{attribute 'TcRpcEnable'}
FUNCTION_BLOCK GetTc3Licenses IMPLEMENTS I_GetTc3Licenses
VAR_INPUT
END_VAR
VAR_OUTPUT
END_VAR
VAR
END_VAR
VAR
    // Internal
    fbGetLicensesEx : FB_GetLicensesEx;
    stAllLicensesInfos : ST_AllLicensesInfos;
    
    _sNetId   : T_AmsNetId;
    
    _fbJson         : FB_JsonSaxWriter;
    _fbJsonDataType : FB_JsonReadWriteDataType;
    
END_VAR
VAR
    stInfoData : ST_LicenseDetailsSmall;
    sReturn : STRING(30_000);
END_VAR


// include: Tc2_Utilities
// Realtime -> Global Max Stack = 2048kb

{attribute 'monitoring' := 'call'}
PROPERTY CountDemoLicenses : UDINT
GET

CountDemoLicenses := stAllLicensesInfos.DemoLicenses.Count;
END_GET
END_PROPERTY

{attribute 'monitoring' := 'call'}
PROPERTY CountFailedLicenses : UDINT
GET

CountFailedLicenses := stAllLicensesInfos.FailedLicenses.Count;
END_GET
END_PROPERTY

{attribute 'monitoring' := 'call'}
PROPERTY CountInvalidLicenses : UDINT
GET

CountInvalidLicenses := stAllLicensesInfos.InvalidLicenses.Count;
END_GET
END_PROPERTY

{attribute 'monitoring' := 'call'}
PROPERTY CountOemLicenses : UDINT
GET

CountOemLicenses := stAllLicensesInfos.OemLicenses.Count;
END_GET
END_PROPERTY

{attribute 'monitoring' := 'call'}
PROPERTY CountPendingLicenses : UDINT
GET

CountPendingLicenses := stAllLicensesInfos.PendingLicenses.Count;
END_GET
END_PROPERTY

{attribute 'monitoring' := 'call'}
PROPERTY CountValidLicenses : UDINT
GET

CountValidLicenses := stAllLicensesInfos.ValidLicenses.Count;
END_GET
END_PROPERTY

METHOD FB_init : BOOL
VAR_INPUT
	bInitRetains : BOOL; // if TRUE, the retain variables are initialized (warm start / cold start)
	bInCopyCode : BOOL;  // if TRUE, the instance afterwards gets moved into the copy code (online change)
    NetId   : T_AmsNetId;
END_VAR

_sNetId := NetId;
END_METHOD

METHOD PUBLIC GetAllLicenses : HRESULT
VAR_INPUT
    bExecute : REFERENCE to BOOL;
END_VAR

IF bExecute THEN
    fbGetLicensesEx(
        bExecute:= bExecute, 
        tTimeout:= , 
        sNetId:= _sNetId, 
        bBusy=> , 
        bError=> , 
        nErrorId=> , 
        nValidLicenses=> stAllLicensesInfos.ValidLicenses.Count, 
        aValidLicenses=> stAllLicensesInfos.ValidLicenses.Info, 
        nPendingLicenses=> stAllLicensesInfos.PendingLicenses.Count, 
        aPendingLicenses=> stAllLicensesInfos.PendingLicenses.Info, 
        nDemoLicenses=> stAllLicensesInfos.DemoLicenses.Count, 
        aDemoLicenses=> stAllLicensesInfos.DemoLicenses.Info, 
        nOemLicenses=> stAllLicensesInfos.OemLicenses.Count, 
        aOemLicenses=> stAllLicensesInfos.OemLicenses.Info, 
        nFailedLicenses=> stAllLicensesInfos.FailedLicenses.Count, 
        aFailedLicenses=> stAllLicensesInfos.FailedLicenses.Info, 
        nInvalidLicenses=> stAllLicensesInfos.InvalidLicenses.Count, 
        aInvalidLicenses=> stAllLicensesInfos.InvalidLicenses.Info);
    
    IF NOT fbGetLicensesEx.bBusy THEN
        bExecute := FALSE;
	END_IF
END_IF
END_METHOD

{attribute 'TcRpcEnable'}
METHOD GetJsonDataLicenses : T_JsonDocLicenseInfoSmall
VAR_INPUT
	LicensesType	: UINT; //E_LicenseType;
END_VAR

CASE LicensesType OF
    E_LicenseType.NoType:
        GetJsonDataLicenses := '';
    E_LicenseType.ValidLicenses:
        GetJsonDataLicenses := JsonDataValidLicenses;
    E_LicenseType.PendingLicenses:
        GetJsonDataLicenses := JsonDataPendingLicenses;
    E_LicenseType.DemoLicenses:
        GetJsonDataLicenses := JsonDataDemoLicenses;
    E_LicenseType.OemLicenses:
        GetJsonDataLicenses := JsonDataOemLicenses;
    E_LicenseType.FailedLicenses:
        GetJsonDataLicenses := JsonDataFailedLicenses;
    E_LicenseType.InvalidLicenses:
        GetJsonDataLicenses := JsonDataInvalidLicenses;
END_CASE
END_METHOD

METHOD PRIVATE GetJsonLicenseDetailSmall : HRESULT
VAR_INPUT
    AdrLicense : XWORD;
    refJsonDoc : REFERENCE TO STRING(30_000);
END_VAR

//Tc2_System.MEMCPY(ADR(stInfoData), ADR(stAllLicensesInfos.ValidLicenses), SIZEOF(stInfoData));
Tc2_System.MEMCPY(ADR(stInfoData), AdrLicense, SIZEOF(stInfoData));

_fbJson.ResetDocument();
_fbJsonDataType.AddJsonValueFromSymbol(_fbJson, 'ST_LicenseDetailsSmall', SIZEOF(stInfoData), ADR(stInfoData));
_fbJson.CopyDocument(sReturn, SIZEOF(sReturn));

refJsonDoc := sReturn;

GetJsonLicenseDetailSmall := S_OK;
END_METHOD

{attribute 'monitoring' := 'call'}
PROPERTY JsonDataDemoLicenses : T_JsonDocLicenseInfoSmall
GET

GetJsonLicenseDetailSmall(ADR(stAllLicensesInfos.DemoLicenses), JsonDataDemoLicenses);
END_GET
END_PROPERTY

{attribute 'monitoring' := 'call'}
PROPERTY JsonDataFailedLicenses : T_JsonDocLicenseInfoSmall
GET

GetJsonLicenseDetailSmall(ADR(stAllLicensesInfos.FailedLicenses), JsonDataFailedLicenses);
END_GET
END_PROPERTY

{attribute 'monitoring' := 'call'}
PROPERTY JsonDataInvalidLicenses : T_JsonDocLicenseInfoSmall
GET

GetJsonLicenseDetailSmall(ADR(stAllLicensesInfos.InvalidLicenses), JsonDataInvalidLicenses);
END_GET
END_PROPERTY

{attribute 'monitoring' := 'call'}
PROPERTY JsonDataOemLicenses : T_JsonDocLicenseInfoSmall
GET

GetJsonLicenseDetailSmall(ADR(stAllLicensesInfos.OemLicenses), JsonDataOemLicenses);
END_GET
END_PROPERTY

{attribute 'monitoring' := 'call'}
PROPERTY JsonDataPendingLicenses : T_JsonDocLicenseInfoSmall
GET

GetJsonLicenseDetailSmall(ADR(stAllLicensesInfos.PendingLicenses), JsonDataPendingLicenses);
END_GET
END_PROPERTY

{attribute 'monitoring' := 'call'}
PROPERTY JsonDataValidLicenses : T_JsonDocLicenseInfoSmall
GET

GetJsonLicenseDetailSmall(ADR(stAllLicensesInfos.ValidLicenses), JsonDataValidLicenses);
END_GET
END_PROPERTY

END_FUNCTION_BLOCK

(* stored: Version 1.1.0.1, ProductVersion 3.1.4024.12
   POU GetTc3Licenses: Id {cfd7b941-6a28-41a7-9746-9138318a2e14}, SpecialFunc None
   Folder Constructor: Id {c24cc863-bf3d-4d9a-b529-7915f882c371}
   Folder ITFs: Id {19d2cf31-f768-4052-88da-48e106115782}
   Folder Methods: Id {4b0d5003-f680-47dd-b2c8-74d43e12db3f}
   Folder Properties: Id {f8f9f002-44e2-418d-aea9-f083ba2761de}
   Folder Privat: Id {b32bcc06-c92e-42cf-8a92-22c168ff433d}
   Folder Public: Id {4337f8a3-7639-41e6-9682-8f6196464927}
   Property CountDemoLicenses: Id {20d6f0c3-fbb7-4f3e-85b1-635f1220d2b6}
   Get Get: Id {13f50410-426c-43bc-8385-eaa7b88a808a}
   Property CountFailedLicenses: Id {af81c4bf-b0b3-483d-b267-47d4e653d0ea}
   Get Get: Id {4f60590c-a6b2-44cc-98bc-d62ee1751929}
   Property CountInvalidLicenses: Id {3aff4063-d7d0-4fd1-b583-691ff5c09428}
   Get Get: Id {b08a783f-f741-4a47-8e92-c7e949fa423e}
   Property CountOemLicenses: Id {afe53d97-8daa-47ab-972f-311227ad3f60}
   Get Get: Id {2fa5a1c5-5546-4352-a9c3-9a03d90b0409}
   Property CountPendingLicenses: Id {eef9b484-cf23-4b7a-a075-2f25bde1b073}
   Get Get: Id {b0ce11ed-382b-469e-aa73-b7fa5a188ff5}
   Property CountValidLicenses: Id {a288c006-012a-40f7-a78e-536a2f09fc17}
   Get Get: Id {fe2beb57-b74b-41be-8b19-cdced04ac034}
   Method FB_init: Id {ade55d3e-d3cb-48c2-9bbd-d9dcfa7526da}
   Method GetAllLicenses: Id {b488a829-a271-42a3-be77-7e8d6d852a83}
   Method GetJsonDataLicenses: Id {5e3341b4-e25b-4a7d-90d0-d8a2857110ab}
   Method GetJsonLicenseDetailSmall: Id {ada069cf-679a-4736-b35a-d44a4bfeb755}
   Property JsonDataDemoLicenses: Id {096ffaee-98b6-48f5-ad1b-af90f111ad2d}
   Get Get: Id {f498a333-1cc8-4603-aadf-972415267fd7}
   Property JsonDataFailedLicenses: Id {cccbb0d0-5fd6-4913-82d3-338099338081}
   Get Get: Id {aab43fac-7643-48a1-ac52-0b266bc94a0e}
   Property JsonDataInvalidLicenses: Id {80bed6d8-0289-4155-9900-c4f715bdb5d1}
   Get Get: Id {2bb90570-6a99-4cb1-850f-f3ba7b683c26}
   Property JsonDataOemLicenses: Id {c5929895-3b69-4a6e-a1d4-3ca48fab32ef}
   Get Get: Id {66d3db60-fdbc-4bb9-bcaa-5eb3914d10ef}
   Property JsonDataPendingLicenses: Id {25d96807-1724-4604-9623-e371bb75103a}
   Get Get: Id {e0cb06a6-246a-46d5-94a6-ac9146b51690}
   Property JsonDataValidLicenses: Id {f5c7c54b-acf4-4d18-8120-6a540700d3b0}
   Get Get: Id {3c32e63a-e260-4c0d-83de-19604e6414e2} *)
